{attribute 'qualified_only'}
{attribute 'strict'}
TYPE MaterialCodes :
(
	NUL,
	
	PAP,
	CAR,
	COR,
	CIP,
	WD
);
END_TYPE

(* stored: Version 1.1.0.1, ProductVersion 3.1.4024.11
   DUT MaterialCodes: Id {216914f2-629c-4a37-941f-9fdd4b398a74} *)
